(* CoDeSys 2.3 export: ERR_RESET_ALL.EXP *)

(* POU Alarm/ERR_RESET_ALL, ST *)
FUNCTION ERR_RESET_ALL : BOOL
VAR_INPUT
	EN: BOOL; (* Сигнал на сброс *)
END_VAR
VAR
	i: INT :=1;
END_VAR
	IF EN THEN
		FOR i := 1 TO _ERR_Nums DO
			ERR_RESET(i);
		END_FOR;
	END_IF;
END_FUNCTION
